Staubli VAL3: detailedStack.pgx

program detailedStack()
  local num i
  local num nTaskStatus
  local num count
  local num j
  local string stack[20]
begin
    //\brief
  //Write detailed stack info to log
  //\var i
  //\var nTaskStatus
  //\var count
  //\var j
  //\var stack
  //
//!brief
  //Write detailed stack info to log
  for i=0 to size(sTaskName)-1
    logMsg("Stack Information for task: "+sTaskName[i])
    nTaskStatus=taskStatus(sTaskName[i])
    // suspend the task
    if nTaskStatus==1
      taskSuspend(sTaskName[i])
    endIf
    // wait until task stopped
    wait(taskStatus(sTaskName[i])!=1)
    // retrieve call stack
    count=$taskCallStack(sTaskName[i],stack)
    // write call stack to log
    for j=0 to count-1
      logMsg(stack[j])
    endFor
    // resume task if it was active when entering this routine
    if nTaskStatus==1
      taskResume(sTaskName[i],0)
    endIf
  endFor
end
